// TIA Portal V18 export
FUNCTION_BLOCK "mot_speed_abs_slowly_accelerated"   // FB67, FBD
{ S7_Optimized_Access := 'TRUE' }
VERSION : 0.1
// stored: AutoNumber true, IsIECCheckEnabled false, IsRetainMemResEnabled false, MemoryReserve 100, SetENOAutomatically false, UDAEnableTagReadback false
   VAR_INPUT
      ALLOWED : Bool;
      set_speed_abs : Real;
      v_absMax : Real;
      t_acc : Real;
   END_VAR
   VAR_OUTPUT
      speed_accelerated_slowly_abs : Real;
   END_VAR
   VAR_TEMP
      cycle_time_s : Real;
      acceleration : Real;
      accleration_per_cycle : Real;
   END_VAR
BEGIN

REGION Network 2 (SCL)
   #cycle_time_s := "_MAIN_DB".CLOCK_S_P_SCAN;
   IF #t_acc > 0 THEN
       #acceleration := #v_absMax / #t_acc;
       #accleration_per_cycle := #acceleration * #cycle_time_s;
       IF NOT #ALLOWED OR #set_speed_abs = 0 THEN
           #speed_accelerated_slowly_abs := #set_speed_abs;
       ELSE
           #speed_accelerated_slowly_abs := LIMIT(MN := 0, IN := #speed_accelerated_slowly_abs + #accleration_per_cycle, MX := #set_speed_abs);
       END_IF;
   ELSE
       #speed_accelerated_slowly_abs := #set_speed_abs;
   END_IF;
END_REGION
END_FUNCTION_BLOCK
